FUNCTION_BLOCK XY_MDLL (* Two-Dimensional Mechanism Model with  Locally Coupled Data+Clock *)
  (* Standard: IEC 61499; Classification: Model; ApplicationDomain: Material Handling; Function: Two-dimensional Motion *)
  (* Version 0.2, 2006-07-07, JHC, Holobloc Inc, Renamed PRESENT to LOADED, moved to top of SENSE. *)
  (* Version 0.1, 2006-06-24, JHC, Holobloc Inc, Renamed HOMEX, ENDX; added HOMEY, ENDY *)
  (* Version 0.0, 2006-06-24, JHC, Holobloc Inc, Adapted from XSLIDE_MDLL. *)
  (* Compiler header: package fb.rt.mach; import fb.rt.mva.*; import fb.rt.net.*; *)
  (* Compiler classdef: public class XY_MDLL extends FBMVCD *)
  (* Compiler Java Sun JDK 1.5.0 *)
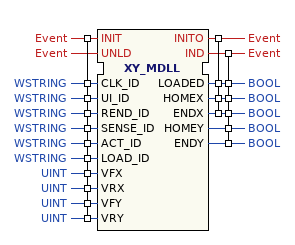
  EVENT_INPUT
    INIT WITH ACT_ID, CLK_ID, UI_ID, SENSE_ID, VFX, VRX, REND_ID, VFY, VRY, LOAD_ID; (* Initialize *)
    UNLD; (* Unload Workpiece *)
  END_EVENT
  EVENT_OUTPUT
    INITO WITH HOMEX, ENDX, LOADED;
    IND WITH HOMEX, ENDX, LOADED, HOMEY, ENDY; (* Sensor Changed *)
  END_EVENT
  VAR_INPUT
    CLK_ID : WSTRING := "SIM_CLK"; (* Simulation clock channel ID *)
    UI_ID : WSTRING; (* User input channel ID from View *)
    REND_ID : WSTRING; (* Local Channel ID for Rendering Data *)
    SENSE_ID : WSTRING; (* Sensor data channel ID to Controller *)
    ACT_ID : WSTRING; (* Actuator data channel ID from Controller *)
    LOAD_ID : WSTRING; (* Workpiece loading data channel ID from Model *)
    VFX : UINT := 10; (* x-axis Forward speed in % Full Scale per CLK event *)
    VRX : UINT := 10; (* x-axis Reverse speed in %FS per CLK event *)
    VFY : UINT := 10; (* y-axis Forward speed in % Full Scale per CLK event *)
    VRY : UINT := 10; (* y-axis Reverse speed in %FS per CLK event *)
  END_VAR
  VAR_OUTPUT
    LOADED : BOOL; (* Workpiece Present *)
    HOMEX : BOOL := 1; (* x-axis at HOME position *)
    ENDX : BOOL; (* x-axis at END position *)
    HOMEY : BOOL := 1; (* y-axis at HOME position *)
    ENDY : BOOL; (* y-axis at END position *)
  END_VAR
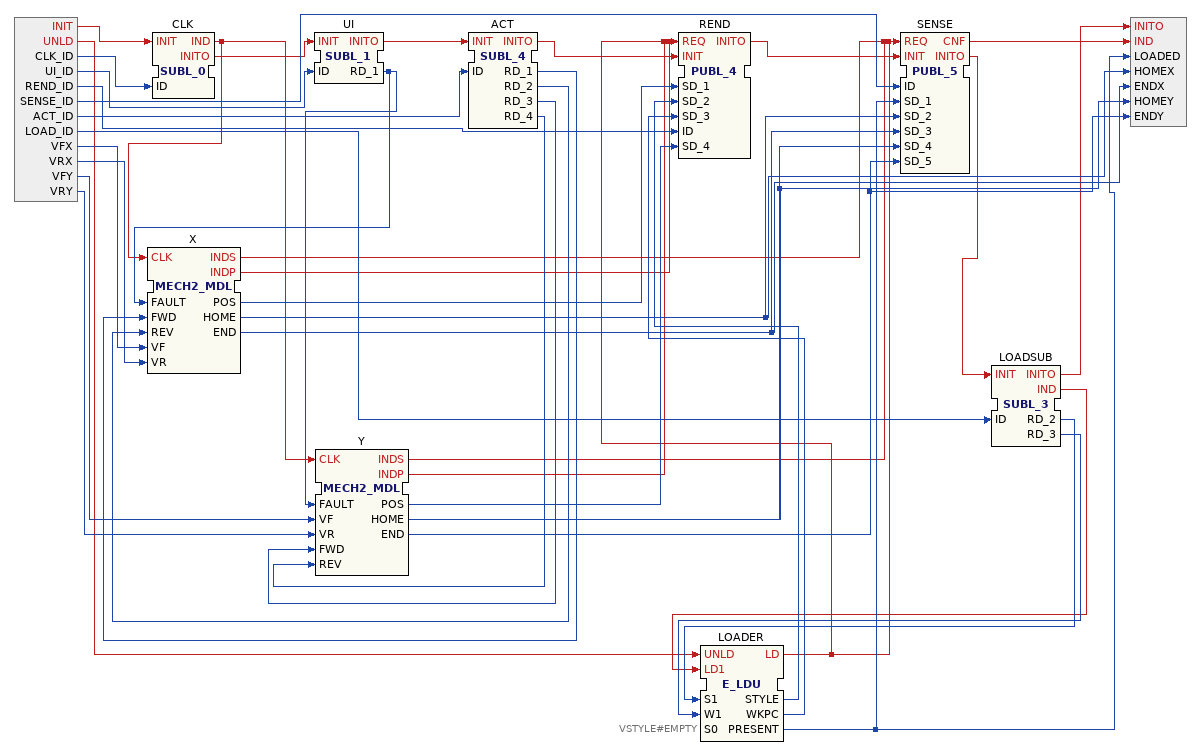
  FBS
    X : MECH2_MDL;
    UI : SUBL_1;
    CLK : SUBL_0;
    ACT : SUBL_4;
    SENSE : PUBL_5;
    REND : PUBL_4;
    LOADER : E_LDU(S0 := VSTYLE#EMPTY);
    Y : MECH2_MDL;
    LOADSUB : SUBL_3; (* Subscriber for Load Channel *)
  END_FBS
  EVENT_CONNECTIONS
    CLK.IND TO X.CLK;
    INIT TO CLK.INIT;
    X.INDS TO SENSE.REQ;
    LOADER.LD TO REND.REQ;
    X.INDP TO REND.REQ;
    UNLD TO LOADER.UNLD;
    LOADER.LD TO SENSE.REQ;
    SENSE.CNF TO IND;
    Y.INDS TO SENSE.REQ;
    CLK.IND TO Y.CLK;
    CLK.INITO TO UI.INIT;
    UI.INITO TO ACT.INIT;
    ACT.INITO TO REND.INIT;
    REND.INITO TO SENSE.INIT;
    SENSE.INITO TO LOADSUB.INIT;
    LOADSUB.INITO TO INITO;
    LOADSUB.IND TO LOADER.LD1;
    Y.INDP TO REND.REQ;
  END_CONNECTIONS
  DATA_CONNECTIONS
    UI.RD_1 TO X.FAULT;
    CLK_ID TO CLK.ID;
    UI_ID TO UI.ID;
    ACT_ID TO ACT.ID;
    ACT.RD_1 TO X.FWD;
    ACT.RD_2 TO X.REV;
    SENSE_ID TO SENSE.ID;
    VFX TO X.VF;
    VRX TO X.VR;
    X.POS TO REND.SD_1;
    LOADER.STYLE TO REND.SD_2;
    LOADER.WKPC TO REND.SD_3;
    REND_ID TO REND.ID;
    Y.POS TO REND.SD_4;
    UI.RD_1 TO Y.FAULT;
    VFY TO Y.VF;
    VRY TO Y.VR;
    ACT.RD_3 TO Y.FWD;
    LOADSUB.RD_2 TO LOADER.S1;
    LOADSUB.RD_3 TO LOADER.W1;
    LOAD_ID TO LOADSUB.ID;
    ACT.RD_4 TO Y.REV;
    LOADER.PRESENT TO SENSE.SD_1;
    X.HOME TO SENSE.SD_2;
    X.END TO SENSE.SD_3;
    Y.HOME TO SENSE.SD_4;
    Y.END TO SENSE.SD_5;
    X.HOME TO HOMEX;
    X.END TO ENDX;
    Y.HOME TO HOMEY;
    Y.END TO ENDY;
    LOADER.PRESENT TO LOADED;
  END_CONNECTIONS
END_FUNCTION_BLOCK
